// TIA Portal V20 export
TYPE "AnalogInDataPLC_DT"
   STRUCT
      LimitUp { ExternalAccessible := 'False'; ExternalVisible := 'False'; ExternalWritable := 'False'} : Real;   // Limit up real value
      LimitDown { ExternalAccessible := 'False'; ExternalVisible := 'False'; ExternalWritable := 'False'} : Real;   // Limit down real value
      TypeProbe { ExternalAccessible := 'False'; ExternalVisible := 'False'; ExternalWritable := 'False'} : Int;   // 0 : PT100, 1 : PT1000, 2 : 0-10V, 3: -10+10V, 4 : RES600, 5 : SL5201 (0-10V), 6 : PTC
      DelayAlarmMin : Time;
      DelayWarningMin : Time;
      DelayWarningMax : Time;
      DelayAlarmMax : Time;
      EnableAlarmMin : Bool;
      EnableWarningMin : Bool;
      EnableWarningMax : Bool;
      EnableAlarmMax : Bool;
      BadPartOnFixture { ExternalVisible := 'False'} : Bool;
   END_STRUCT;
END_TYPE
